{attribute 'qualified_only'}
VAR_GLOBAL
	{attribute 'OPC.UA.DA' := '1'}
	fTE         : ARRAY [1..19] OF REAL;
	{attribute 'OPC.UA.DA' := '1'}
    bHV AT %Q*  : ARRAY [1..11] OF BOOL;
	{attribute 'OPC.UA.DA' := '1'}
    bFan AT %Q*  : BOOL;
	{attribute 'OPC.UA.DA' := '1'}
    bST         : BOOL;
	{attribute 'OPC.UA.DA' := '1'}
	stP1		: GrundfosMagna3;
	{attribute 'OPC.UA.DA' := '1'}
	stP2		: GrundfosMagna3;
	{attribute 'OPC.UA.DA' := '1'}
	stFeeder	: ATV212;
	{attribute 'OPC.UA.DA' := '1'}
	bLoadTank1	: BOOL := TRUE;
	{attribute 'OPC.UA.DA' := '1'}
	bLoadTank2	: BOOL := TRUE;
	{attribute 'OPC.UA.DA' := '1'}
	bLoadTank3	: BOOL := TRUE;
END_VAR

(* stored: Version 1.1.0.1, ProductVersion 3.1.4022.18
   GVL GVL: Id {884c114f-e978-4949-b759-3e84d5a1e2f7} *)
